TYPE ST_SolventsSettings :
STRUCT
	sSolventName	: STRING(80); 	// The name of the solvent inserted on the settings screen
	rDensity		: LREAL;		// The density of this solvent
END_STRUCT
END_TYPE

(* stored: Version 1.1.0.1, ProductVersion 3.1.4024.15
   DUT ST_SolventsSettings: Id {d654a11b-cae7-4542-ba7f-91395eb04e38} *)
